TYPE ST_HartingIO_set :
STRUCT
	w_SwitchControlSignals		: 	WORD; // control signals for output contact
	r_manualAnalogOutput		: 	REAL; // 0 - 100%
	r_gensetAnalogOutput		: 	REAL; // 0 - 100%
	r_HpuAnalogOutput			: 	REAL; // 0 - 100%
END_STRUCT
END_TYPE

(* stored: Version 1.1.0.1, ProductVersion 3.1.4026.18
   DUT ST_HartingIO_set: Id {7d510f51-5bd1-4664-a84d-5af18a4a4b86} *)
